Fanuc KAREL source: kb00005.KL

-- PROVISIONAL review KL for V940-1; original PC SHA256 308f7910ae7e4ab86d5a0814e0832007b99b52c55befd16d4fed4b7fd10b6131
-- Incomplete behavior may be omitted. Consult companion uncertainty JSON. Do not deploy.
PROGRAM KB00005
%NOLOCKGROUP
BEGIN
  -- V9_ZERO_TABLE_METADATA_HINT layout=0002_ascii; no indexed target words; source/name/runtime held
  -- UNRESOLVED_PC offsets 5-14; opcodes 3F,75
  -- UNRESOLVED_PC offsets 19-28; opcodes 3F,75
  -- UNRESOLVED_PC offsets 33-42; opcodes 3F,75
  -- UNRESOLVED_PC offsets 47-54; opcodes 9D,23
  -- UNRESOLVED_PC offsets 59-66; opcodes 9D,23
  -- UNRESOLVED_PC offsets 71-111; opcodes 27,22,2A,22,2A,22,2A,22,22,31
  -- UNRESOLVED_PC offsets 116-120; opcodes 7F
END KB00005
